FUNCTION_BLOCK GetInstancePathAndName (* Function block to retrieve instance path and instance name from the runtime *)
  (* Description: Copyright (c) 2024 Primetals Technologies Austria GmbH This program and the accompanying materials are made available under the terms of the Eclipse Public License 2.0 which is available at https://www.eclipse.org/legal/epl-2.0/ SPDX-License-Identifier: EPL-2.0 *)
  (* Version 1.0, 2024-04-10, Ernst Blecha, Primetals Technologies Austria GmbH *)
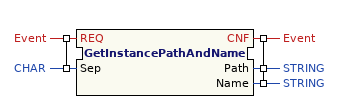
  EVENT_INPUT
    REQ WITH Sep; (* Service Request *)
  END_EVENT
  EVENT_OUTPUT
    CNF WITH Path, Name; (* Confirmation of Requested Service *)
  END_EVENT
  VAR_INPUT
    Sep : CHAR := '/'; (* Separator character for the output path generated by this FB *)
  END_VAR
  VAR_OUTPUT
    Path : STRING; (* Instance path of this FB *)
    Name : STRING; (* Instance name of this FB *)
  END_VAR
END_FUNCTION_BLOCK
